// Mitsubishi GX Works2 project: 0703-공개문제20카운터실패   PLC: Q02/Q02H

PROGRAM MAIN
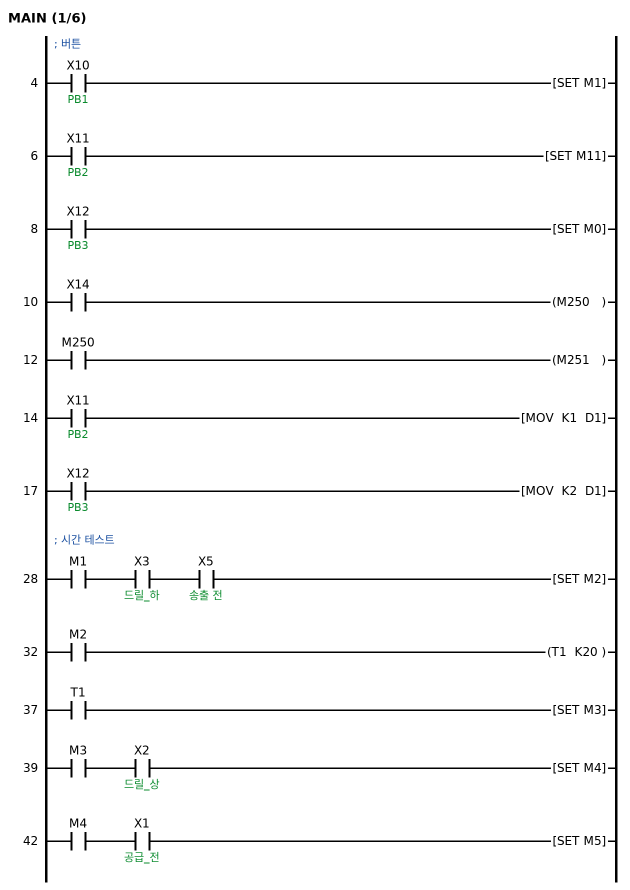
; 버튼
4     LD      X10  ; PB1
      SET     M1
6     LD      X11  ; PB2
      SET     M11
8     LD      X12  ; PB3
      SET     M0
10    LD      X14
      OUT     M250
12    LD      M250
      OUT     M251
14    LD      X11  ; PB2
      MOV     K1 D1
17    LD      X12  ; PB3
      MOV     K2 D1
; 시간 테스트
28    LD      M1
      AND     X3  ; 드릴_하
      AND     X5  ; 송출 전
      SET     M2
32    LD      M2
      OUT     T1 K20
37    LD      T1
      SET     M3
39    LD      M3
      AND     X2  ; 드릴_상
      SET     M4
42    LD      M4
      AND     X1  ; 공급_전
      SET     M5
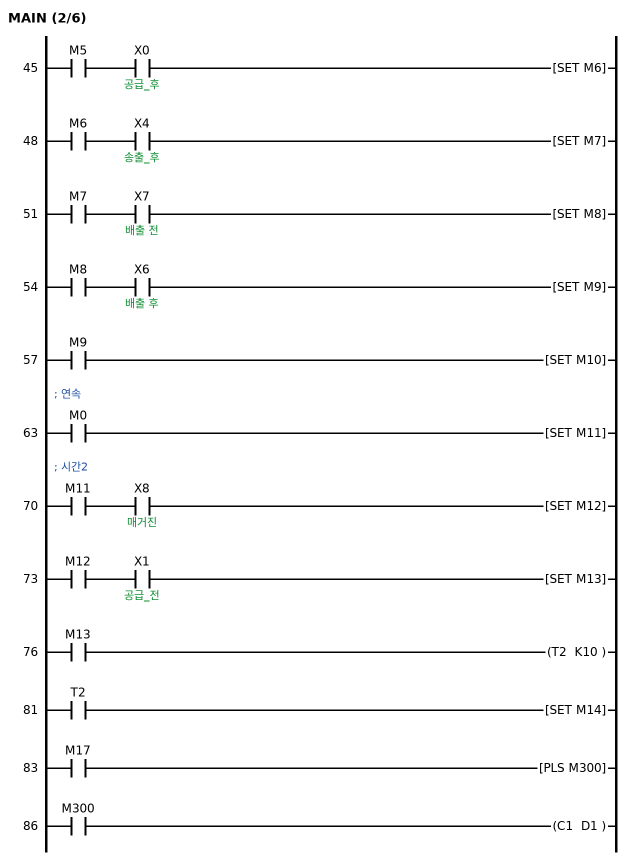
45    LD      M5
      AND     X0  ; 공급_후
      SET     M6
48    LD      M6
      AND     X4  ; 송출_후
      SET     M7
51    LD      M7
      AND     X7  ; 배출 전
      SET     M8
54    LD      M8
      AND     X6  ; 배출 후
      SET     M9
57    LD      M9
      SET     M10
; 연속
63    LD      M0
      SET     M11
; 시간2
70    LD      M11
      AND     X8  ; 매거진
      SET     M12
73    LD      M12
      AND     X1  ; 공급_전
      SET     M13
76    LD      M13
      OUT     T2 K10
81    LD      T2
      SET     M14
83    LD      M17
      PLS     M300
86    LD      M300
      OUT     C1 D1
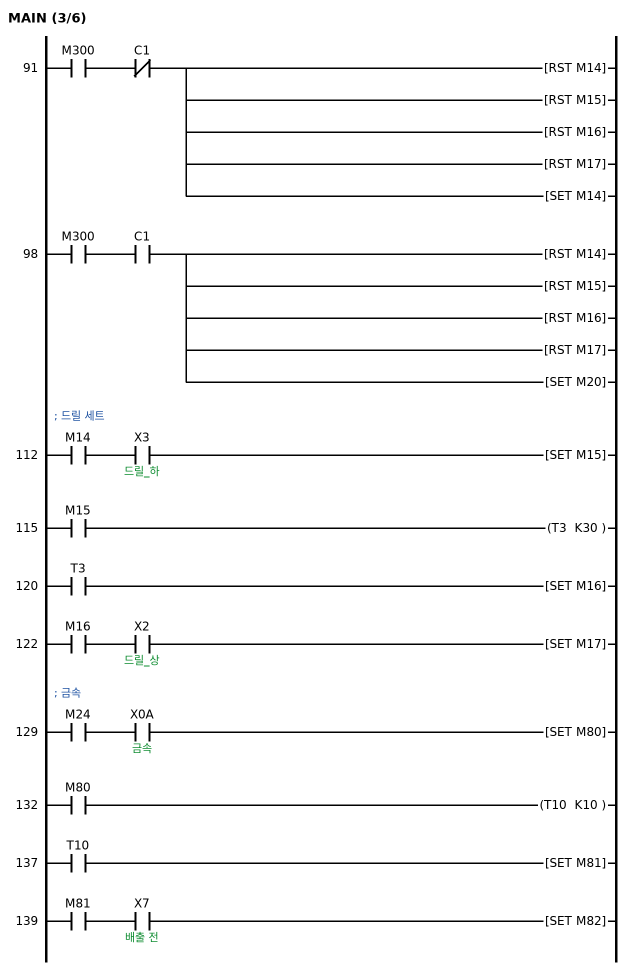
91    LD      M300
      ANI     C1
      RST     M14
      RST     M15
      RST     M16
      RST     M17
      SET     M14
98    LD      M300
      AND     C1
      RST     M14
      RST     M15
      RST     M16
      RST     M17
      SET     M20
; 드릴 세트
112   LD      M14
      AND     X3  ; 드릴_하
      SET     M15
115   LD      M15
      OUT     T3 K30
120   LD      T3
      SET     M16
122   LD      M16
      AND     X2  ; 드릴_상
      SET     M17
; 금속
129   LD      M24
      AND     X0A  ; 금속
      SET     M80
132   LD      M80
      OUT     T10 K10
137   LD      T10
      SET     M81
139   LD      M81
      AND     X7  ; 배출 전
      SET     M82
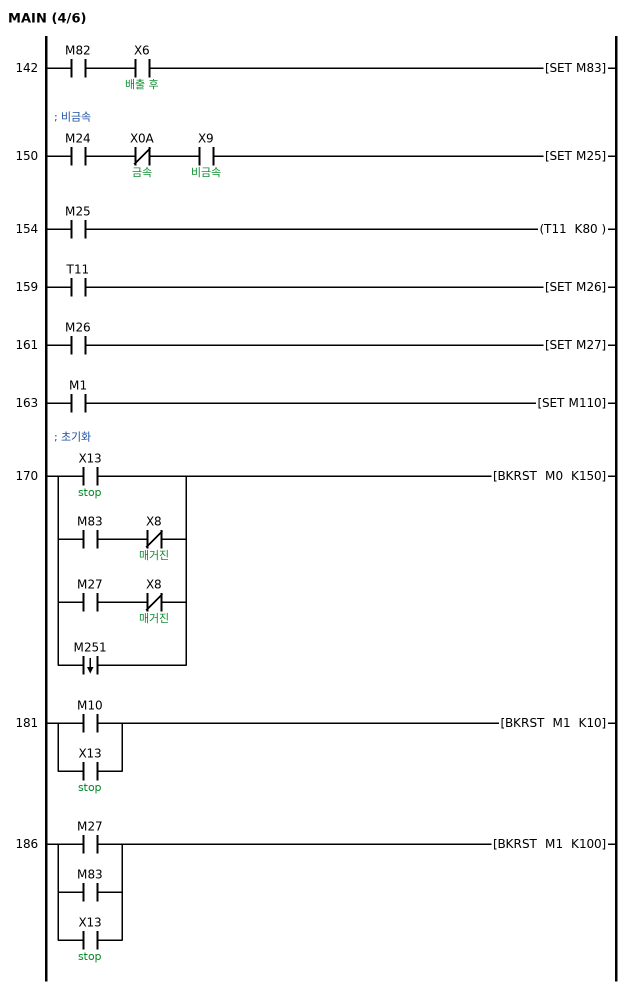
142   LD      M82
      AND     X6  ; 배출 후
      SET     M83
; 비금속
150   LD      M24
      ANI     X0A  ; 금속
      AND     X9  ; 비금속
      SET     M25
154   LD      M25
      OUT     T11 K80
159   LD      T11
      SET     M26
161   LD      M26
      SET     M27
163   LD      M1
      SET     M110
; 초기화
170   LD      X13  ; stop
      LD      M83
      ANI     X8  ; 매거진
      ORB
      LD      M27
      ANI     X8  ; 매거진
      ORB
      ORF     M251
      BKRST   M0 K150
181   LD      M10
      OR      X13  ; stop
      BKRST   M1 K10
186   LD      M27
      OR      M83
      OR      X13  ; stop
      BKRST   M1 K100
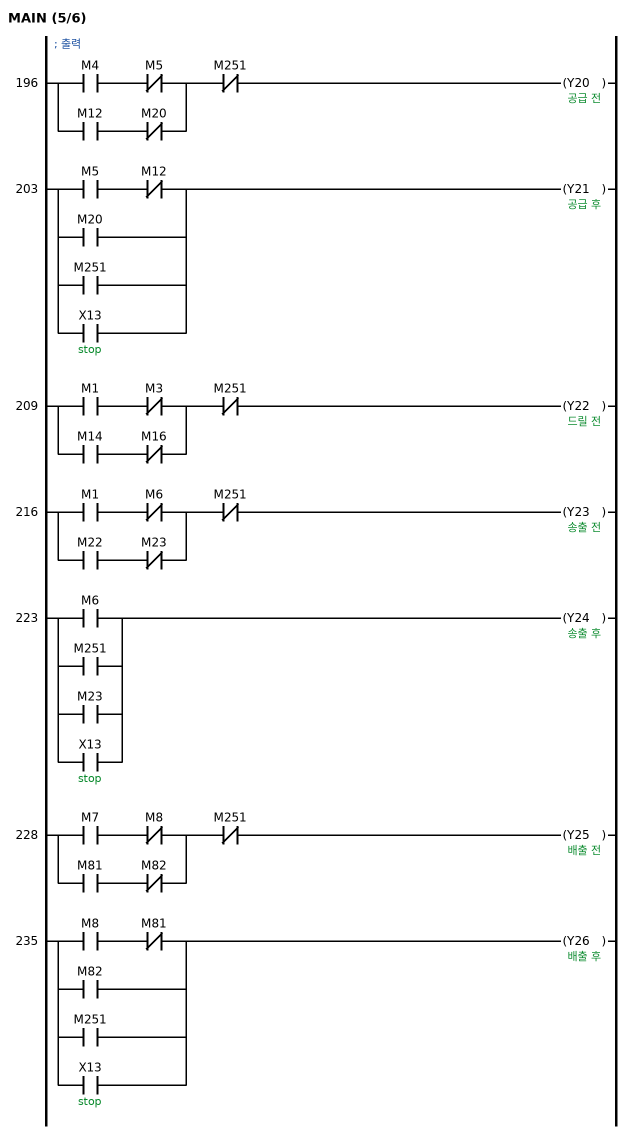
; 출력
196   LD      M4
      ANI     M5
      LD      M12
      ANI     M20
      ORB
      ANI     M251
      OUT     Y20  ; 공급 전
203   LD      M5
      ANI     M12
      OR      M20
      OR      M251
      OR      X13  ; stop
      OUT     Y21  ; 공급 후
209   LD      M1
      ANI     M3
      LD      M14
      ANI     M16
      ORB
      ANI     M251
      OUT     Y22  ; 드릴 전
216   LD      M1
      ANI     M6
      LD      M22
      ANI     M23
      ORB
      ANI     M251
      OUT     Y23  ; 송출 전
223   LD      M6
      OR      M251
      OR      M23
      OR      X13  ; stop
      OUT     Y24  ; 송출 후
228   LD      M7
      ANI     M8
      LD      M81
      ANI     M82
      ORB
      ANI     M251
      OUT     Y25  ; 배출 전
235   LD      M8
      ANI     M81
      OR      M82
      OR      M251
      OR      X13  ; stop
      OUT     Y26  ; 배출 후
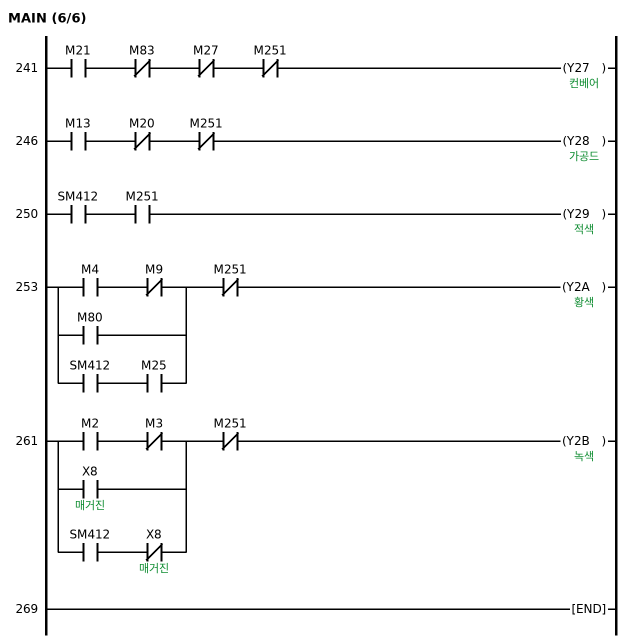
241   LD      M21
      ANI     M83
      ANI     M27
      ANI     M251
      OUT     Y27  ; 컨베어
246   LD      M13
      ANI     M20
      ANI     M251
      OUT     Y28  ; 가공드
250   LD      SM412
      AND     M251
      OUT     Y29  ; 적색
253   LD      M4
      ANI     M9
      OR      M80
      LD      SM412
      AND     M25
      ORB
      ANI     M251
      OUT     Y2A  ; 황색
261   LD      M2
      ANI     M3
      OR      X8  ; 매거진
      LD      SM412
      ANI     X8  ; 매거진
      ORB
      ANI     M251
      OUT     Y2B  ; 녹색
269   END
END_PROGRAM

PROGRAM MAIN1
0     END
END_PROGRAM
